PROGRAM Axis01_Auto
VAR
//System_Bit
	Always_ON	:	BOOL	:=TRUE	;//상시 ON 
	Always_OFF	:	BOOL	:=FALSE	;//상시 OFF
END_VAR

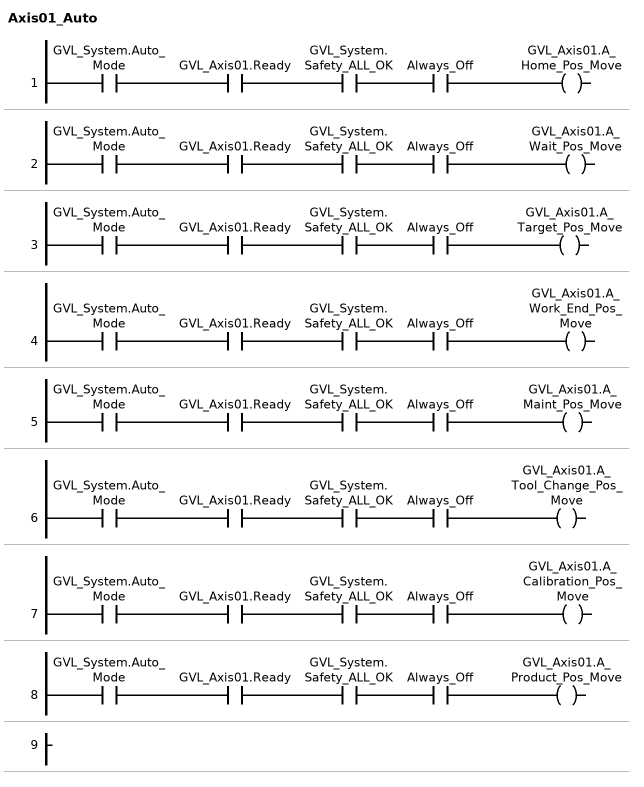
// NETWORK 1
GVL_Axis01.A_Home_Pos_Move := GVL_System.Auto_Mode AND GVL_Axis01.Ready AND GVL_System.Safety_ALL_OK AND Always_Off;

// NETWORK 2
GVL_Axis01.A_Wait_Pos_Move := GVL_System.Auto_Mode AND GVL_Axis01.Ready AND GVL_System.Safety_ALL_OK AND Always_Off;

// NETWORK 3
GVL_Axis01.A_Target_Pos_Move := GVL_System.Auto_Mode AND GVL_Axis01.Ready AND GVL_System.Safety_ALL_OK AND Always_Off;

// NETWORK 4
GVL_Axis01.A_Work_End_Pos_Move := GVL_System.Auto_Mode AND GVL_Axis01.Ready AND GVL_System.Safety_ALL_OK AND Always_Off;

// NETWORK 5
GVL_Axis01.A_Maint_Pos_Move := GVL_System.Auto_Mode AND GVL_Axis01.Ready AND GVL_System.Safety_ALL_OK AND Always_Off;

// NETWORK 6
GVL_Axis01.A_Tool_Change_Pos_Move := GVL_System.Auto_Mode AND GVL_Axis01.Ready AND GVL_System.Safety_ALL_OK AND Always_Off;

// NETWORK 7
GVL_Axis01.A_Calibration_Pos_Move := GVL_System.Auto_Mode AND GVL_Axis01.Ready AND GVL_System.Safety_ALL_OK AND Always_Off;

// NETWORK 8
GVL_Axis01.A_Product_Pos_Move := GVL_System.Auto_Mode AND GVL_Axis01.Ready AND GVL_System.Safety_ALL_OK AND Always_Off;

// NETWORK 9

END_PROGRAM

(* stored: Version 1.1.0.1, ProductVersion 3.1.4024.15
   POU Axis01_Auto: Id {ddfc8f39-dd17-40fe-a351-b7f2ce3decf3}, SpecialFunc None *)
